(* IEC 61131-3 sources: POMIRTS_lab3/AS/Library_2/vncserv, 2 files *)

(* ---- VncServ.fun ---- *)
(********************************************************************
 * COPYRIGHT (C) BERNECKER + RAINER, AUSTRIA, A-5142 EGGELSBERG
 ********************************************************************
 * Library: VncServ
 * File: VncServ.fun
 * Created: 11.11.2003
 ********************************************************************
 * Functions and function blocks of library VncServ
 ********************************************************************)
FUNCTION VNC_Start : UINT (*start vnc server *)
	VAR_INPUT
		Resolution	:USINT; (*screen resolution*)
		Port	:UINT; (*port*)
		RefreshTime	:USINT; (*refresh time in ms*)
		Interpreter	:STRING[80]; (*name of visualization*)
		TargetHW	:USINT; (*type of hardware*)
	END_VAR
END_FUNCTION
FUNCTION VNC_Stop : UINT (*stop vnc server *)
END_FUNCTION
FUNCTION VNC_Quit : UINT (*shut down vnc server *)
END_FUNCTION

(* ---- VncServ.var ---- *)
(********************************************************************
 * COPYRIGHT (C) BERNECKER + RAINER, AUSTRIA, A-5142 EGGELSBERG
 ********************************************************************
 * Library: VncServ
 * File: VncServ.var
 * Created: 11.11.2003
 ********************************************************************
 * Constants of library VncServ
 ********************************************************************)
VAR CONSTANT
	RES1024x768	: USINT	:= 4;
	RES800x600	: USINT	:= 3;
	RES640x480	: USINT	:= 1;
	RES320x240	: USINT	:= 2;
	IMMEDIATE	: USINT	:= 2;
	VERYHIGH	: USINT	:= 4;
	IPCXXXX	: USINT	:= 0;
	PPXXX	: USINT	:= 1;
	HIGH	: USINT	:= 3;
	LOW	: USINT	:= 1;
END_VAR
